// TIA Portal V21 export
DATA_BLOCK "FillWfi"   // DB302
AUTHOR : PRECISE
FAMILY : PRECISE
// stored: AutoNumber false, InstanceOfName FB301, InstanceOfType FB
"FB301"
   // VAR_INPUT
   //    Enable : Bool;
   //    Disable : Bool;
   //    Fault : Bool;
   //    SecPulse : Bool;
   //    AlwaysTrue : Bool;
   //    StartConfirmationPopupSel : Bool;
   //    EndConfirmationPopupSel : Bool;
   //    FillModeSel : Int;
   //    FillMethodSel : Int;
   //    FillTimeBaseSel : Bool;
   //    FillLineSel : Int;
   //    InitialDrainSel : Bool := 1;
   //    SBIPulsingSel : Bool;
   //    FinalVolumeMakeupSel : Bool;
   //    PurgingSel : Bool;
   //    UtilitySel : Bool;
   //    FillQuantity : Real := 10.0;
   //    FillTimeMin : Int;
   //    FillTimeSec : Int;
   //    ActualQuantity : Real;
   //    InflightQuantity : Real;
   //    ZDVDelay : Int;
   //    InitialDrainDelay : Int := 20;
   //    PurgingTime : Int;
   //    SBIOnTime : Int;
   //    SBIOffTime : Int;
   //    SetQuantitytoStartPulsing : Real;
   //    FillQuantityTolerance : Real;
   //    PrintInetrval : Int;
   // END_VAR
   // VAR_OUTPUT
   //    PWZDV : Bool;
   //    WFIZDV : Bool;
   //    PWLineValves : Bool;
   //    WFILineValves : Bool;
   //    InitialDrainValves : Bool;
   //    SBIValve : Bool;
   //    JTubeValve : Bool;
   //    AirInletValve : Bool;
   //    StartConfirmationPopup : Bool;
   //    EndConfirmationPopup : Bool;
   //    ManualPopup : Bool;
   //    AlarmFillQuantityExeeded : Bool;
   //    FillTimeMinPV : DInt;
   //    FillTimeSecPV : DInt;
   //    PrintTrigger : Bool;
   //    PrintWord : Int;
   //    PrintStatus : String[50];
   // END_VAR
   // VAR_IN_OUT
   //    Start : Bool;
   //    Stop : Bool;
   //    Reset : Bool;
   //    StartConfirmationAck : Bool;
   //    EndConfirmationAck : Bool;
   //    ManualAck : Bool;
   //    AlarmAck : Bool;
   //    SpareBtn1 : Bool;
   //    Running : Bool;
   //    Selected : Bool;
   //    Paused : Bool;
   //    StartConfirmationPopupTemp : Bool;
   //    EndConfirmationPopupTemp : Bool;
   //    ManualPopupTemp : Bool;
   //    InitialDrainDelayStarted : Bool;
   //    InitialDrainDelayOver : Bool;
   //    FillStarted : Bool;
   //    FillOver : Bool;
   //    FillOverTemp : Bool;
   //    InitialDrainDelayPV : Int;
   //    ActualFillQuantityCalc : Real;
   //    ActualFillQuantity : Real;
   //    PulsingStartWeight : Real;
   //    PurgingTimePV : Int;
   //    FillQuantityToleranceCalc : Real;
   //    VesselMaxWeight : Real := 13000.0;
   //    ResetBatchTimer : Bool;
   // END_VAR
   // VAR
   //    ValveOnDelayPV : Int;
   //    ValveOffDelayPV : Int;
   //    PrintTriggerTemp : Bool;
   //    RE1 : Bool;
   //    RE2 : Bool;
   //    RE3 : Bool;
   //    RE4 : Bool;
   //    RE5 : Bool;
   //    RE6 : Bool;
   //    RE7 : Bool;
   //    FillTimer { S7_SetPoint := 'True'} : "FB101";
   //    SBIPulsing { S7_SetPoint := 'True'} : "FB102";
   //    PrintTriggerResetTimer { S7_SetPoint := 'True'} : TON_TIME;
   //    BtnResetTimer { S7_SetPoint := 'True'} : TON_TIME;
   //    IEC_Counter_0_Instance { S7_SetPoint := 'True'} : CTU_INT;
   // END_VAR
BEGIN
END_DATA_BLOCK
